PROGRAM PIST_CYCLE
VAR
	bFirstRun:BOOL:=FALSE;
	counter :INT;
END_VAR


//IF NOT bFirstRun THEN
//	FOR counter:=1 TO iNUMBER_OF_PISTONS BY 1 DO
//		fbPist[counter].bInit:=1;
//	END_FOR;
//bFirstRun:=TRUE;
//END_IF
 

grp1();

ACTION grp1:
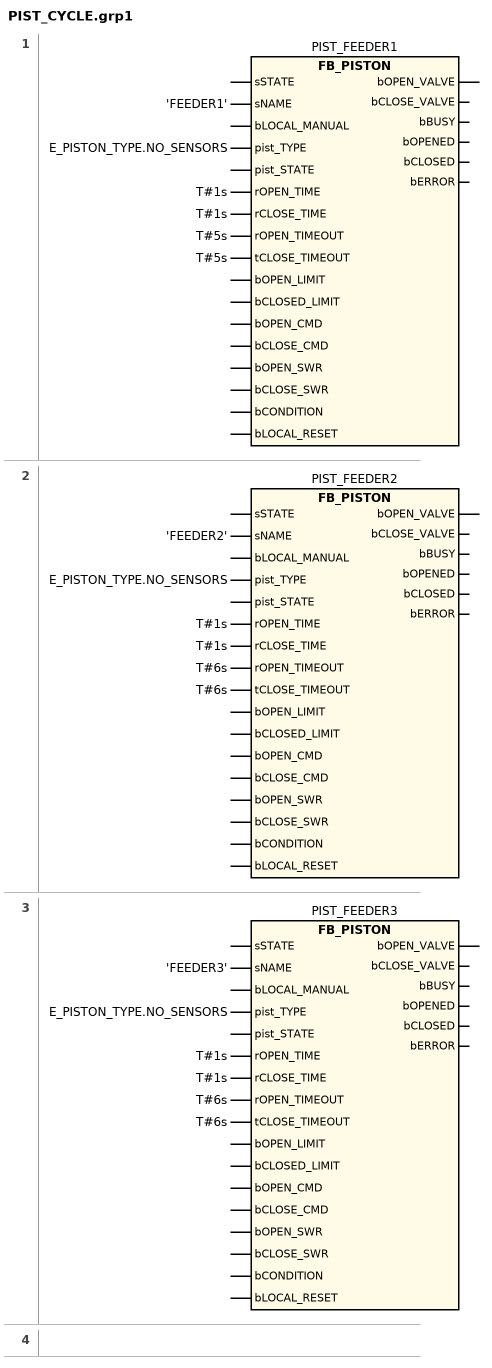
// NETWORK 1
PIST_FEEDER1(
    sNAME := 'FEEDER1',
    pist_TYPE := E_PISTON_TYPE.NO_SENSORS,
    rOPEN_TIME := T#1s,
    rCLOSE_TIME := T#1s,
    rOPEN_TIMEOUT := T#5s,
    tCLOSE_TIMEOUT := T#5s); // FB_PISTON

// NETWORK 2
PIST_FEEDER2(
    sNAME := 'FEEDER2',
    pist_TYPE := E_PISTON_TYPE.NO_SENSORS,
    rOPEN_TIME := T#1s,
    rCLOSE_TIME := T#1s,
    rOPEN_TIMEOUT := T#6s,
    tCLOSE_TIMEOUT := T#6s); // FB_PISTON

// NETWORK 3
PIST_FEEDER3(
    sNAME := 'FEEDER3',
    pist_TYPE := E_PISTON_TYPE.NO_SENSORS,
    rOPEN_TIME := T#1s,
    rCLOSE_TIME := T#1s,
    rOPEN_TIMEOUT := T#6s,
    tCLOSE_TIMEOUT := T#6s); // FB_PISTON

// NETWORK 4
END_ACTION

END_PROGRAM

(* stored: Version 1.1.0.1, ProductVersion 3.1.4024.12
   POU PIST_CYCLE: Id {b09e4efb-d7ec-45c6-bc50-8222237b347f}, SpecialFunc None
   Action grp1: Id {b6db8f46-a5cd-4841-b2f4-af5cb236d344} *)
